FUNCTION_BLOCK FB_Roboter_Logik
VAR_INPUT
	bEnable :BOOL;
	bExecute :BOOL;

	pPositionX :REAL;
	bRefmin_X :BOOL;
	bRefmax_X :BOOL;
	
	pPositionY :REAL;
	bRefmin_Y :BOOL;
	bRefmax_Y :BOOL;
	
	pPositionZ :REAL;
	bRefmin_Z :BOOL;
	bRefmax_Z :BOOL;
	
	
	
	
END_VAR
VAR_OUTPUT
	bBreak :BOOL;
	
	
	eState :eBetriebszustand;
	
END_VAR
VAR
	fb_Roboter_Axis_X : FB_Roboter_Axis;
	fb_Roboter_Axis_Y : FB_Roboter_Axis;
	fb_Roboter_Axis_Z : FB_Roboter_Axis;
	//fb_Roboter_Gripper : FB_Roboter_Axis;
	
	nState :INT;
END_VAR

//soft limits bei Achse selbst für realen Betrieb einstellen 

fb_Roboter_Axis_X(
	bEnable:= , 
	bExecute:= , 
	rPosition:= , 
	bRefSens:= bRefmin_X, 
	eState=> , 
	ax:= IFC_HW.ax_ManX);
fb_Roboter_Axis_Y(
	bEnable:= , 
	bExecute:= , 
	rPosition:= , 
	bRefSens:= bRefmin_Y, 
	eState=> , 
	ax:= IFC_HW.ax_ManY);
fb_Roboter_Axis_Z(
	bEnable:= , 
	bExecute:= , 
	rPosition:= , 
	bRefSens:= bRefmin_Z, 
	eState=> , 
	ax:= IFC_HW.ax_ManZ);

IF NOT bEnable THEN
	nState :=0;
END_IF

CASE nState OF
	0: //off
	eState := eBetriebszustand.Off;
	
	IF bEnable THEN
		nstate :=1;
	END_IF
	
	1: //init
	eState := eBetriebszustand.Init;
	fb_Roboter_Axis_X.bEnable := TRUE;
	fb_Roboter_Axis_Y.bEnable := TRUE;
	fb_Roboter_Axis_Z.bEnable := TRUE;
	
	IF (fb_Roboter_Axis_X.eState = eBetriebszustand.Ready) AND (fb_Roboter_Axis_Y.eState = eBetriebszustand.Ready) AND (fb_Roboter_Axis_Z.eState = eBetriebszustand.Ready) THEN 
		nstate :=2;
	END_IF
	
	2: //Ready
	eState := eBetriebszustand.Ready;
	
	IF bExecute THEN 
		nstate :=21;
	END_IF
	
	21: //check z hight
	eState := eBetriebszustand.Production;
	
	IF IFC_HW.ax_ManZ.NcToPlc.ActPos > GVL_PosKinematic.pZoff THEN
		nstate :=22;
	ELSE
		nstate :=23;
	END_IF
	
	22: //Move Z to safe position
	eState := eBetriebszustand.Production;
	
	fb_Roboter_Axis_Z.rPosition :=45;
	fb_Roboter_Axis_Z.bExecute :=TRUE;
	bBreak :=TRUE;
	
	IF fb_Roboter_Axis_Z.eState = eBetriebszustand.Done THEN
		fb_Roboter_Axis_Z.bExecute :=FALSE;
		bBreak :=FALSE;
		nstate :=23;
	END_IF
	
	23: //Move xy
	eState := eBetriebszustand.Production;
	
	fb_Roboter_Axis_X.rPosition :=pPositionX;
	fb_Roboter_Axis_X.bExecute :=TRUE;
	fb_Roboter_Axis_Y.rPosition :=pPositionY;
	fb_Roboter_Axis_Y.bExecute :=TRUE;
	
	IF (fb_Roboter_Axis_X.eState = eBetriebszustand.Done) AND (fb_Roboter_Axis_Y.eState = eBetriebszustand.Done) THEN
		fb_Roboter_Axis_X.bExecute :=FALSE;
		fb_Roboter_Axis_Y.bExecute :=FALSE;
		nstate :=24;
	END_IF
	
	24: //Move Z
	eState := eBetriebszustand.Production;
	
	fb_Roboter_Axis_Z.rPosition :=pPositionZ;
	fb_Roboter_Axis_Z.bExecute :=TRUE;
	bBreak :=TRUE;
	
	IF fb_Roboter_Axis_Z.eState = eBetriebszustand.Done THEN
		fb_Roboter_Axis_Z.bExecute :=FALSE;
		bBreak :=FALSE;
		nstate :=25;
	END_IF
	
	25: //Done
	eState := eBetriebszustand.Done;
	
	IF NOT bExecute THEN
		nstate :=2;
	END_IF
	
	
END_CASE

END_FUNCTION_BLOCK

(* stored: Version 1.1.0.1, ProductVersion 3.1.4024.15
   POU FB_Roboter_Logik: Id {8ba7399c-3ab9-4824-9167-bb4531069ea3}, SpecialFunc None *)
